Yaskawa INFORM job: P_Y.JBI

/JOB
//NAME P_Y
///FOLDERNAME INNE
//POS
///NPOS 7,7,7,0,0,0
///TOOL 0
///POSTYPE PULSE
///PULSE
C00000=31500,-26929,29037,8977,76581,9154
C00001=29973,6708,54635,8524,78236,8810
C00002=18064,49160,98551,5301,73922,5098
C00003=-9873,55162,104950,-4085,71253,-2372
C00004=-23209,27720,74666,-6658,77272,-6751
C00005=-30212,-2525,46736,-8564,78341,-8891
C00006=-26658,-36149,23390,-7663,75763,-7667
BC00000=103636,1063120,678618
BC00001=103636,1063121,678621
BC00002=103636,1063121,678621
BC00003=103636,1063121,678621
BC00004=103636,1063121,678621
BC00005=103636,1063121,678621
BC00006=103636,1063121,678621
EC00000=0,1
EC00001=0,239555
EC00002=0,501510
EC00003=0,974886
EC00004=0,1204752
EC00005=0,1402700
EC00006=0,1659361
//INST
///DATE 2023/10/04 15:13
///ATTR SC,RW
///GROUP1 RB1,BS1
///GROUP2 ST1
NOP
MOVJ C00000 BC00000 VJ=0.78  +MOVJ EC00000 VJ=0.78
MOVJ C00001 BC00001 VJ=0.78  +MOVJ EC00001 VJ=0.78
MOVJ C00002 BC00002 VJ=0.78  +MOVJ EC00002 VJ=0.78
MOVJ C00003 BC00003 VJ=0.78  +MOVJ EC00003 VJ=0.78
MOVJ C00004 BC00004 VJ=0.78  +MOVJ EC00004 VJ=0.78
MOVJ C00005 BC00005 VJ=0.78  +MOVJ EC00005 VJ=0.78
MOVJ C00006 BC00006 VJ=0.78  +MOVJ EC00006 VJ=0.78
END
